	FUNCTION_BLOCK FB 1054
	TITLE =A_2615_MXZ15MA LIFTING SCREW
	//COPYRIGHT:     (C) 2009  BUHLER AG, CH-9240 UZWIL, SWITZERLAND
	//
	//PRODUCT:       WinCoS_BIW01_09
	//
	//TITLE:         LIFTING SCREW
	//
	//--------------------------------------------------------------------------------
	//
	//IDENT:         AUTHOR:             DEPT:                             DATE:
	//
	//P01_FB1054.1.0 K.Renz              CSB41                             13.Jan.2010
	//               1st Release
	//
	//--------------------------------------------------------------------------------
	//
	//PURPOSE:
	//
	//MANUAL :
	//
	//RESTRICTIONS:
	//
	//--------------------------------------------------------------------------------
	AUTHOR  : KR
	FAMILY  : USW
	VERSION : 0.0


	VAR
	         Ma :  UDT 20500  ;  // Machine
	         A_2615_BTT15 : FB14;  // Mon1: DigInpCont
	         A_2615_BSA17 : FB14;  // Mon2: DigInpCont
	         Mon3  : FB14  ;  // spare
	         Mon4  : FB14 ;  // spare
	         Mon5  : FB14 ;   // spare
	         Mon6  : FB14 ;   // spare
	         A_2615_MXZ15 : FB12; // Motor: Motor
	END_VAR

	BEGIN
	NETWORK
	TITLE =Call SSW
	   UC  FB50
	END_FUNCTION_BLOCK
